GVL_MaintainLaser.q_bShutoffLatch := GVL_MaintainLaser.q_bShutoffLatch
	OR GVL_MaintainLaser.i_bShutoff
	OR NOT bSwitchboxStatusOk;
		
FOR nIter := 1 TO GVL_TransportTubes.NUM_TRANSPORT_TUBES DO
	eTT := GVL_TransportTubes.aTubes[nIter];
	fbTT REF= F_GetTransportTube(eTT);
	
	(* Disable Laser Ok signal if transport tube or switchbox is in bad state *)
	IF GVL_MaintainLaser.q_bShutoffLatch
	OR NOT F_VerifyTransportTubeStatuses(stExpStatus := stExpTTStatus,
		eTransportTube := eTT,
		stStatusOp := stTTOp, 
		bEnforce := FALSE)
	THEN // System status is not ok. Disable laser Ok signal
		fbTT.M_SetLaserOk(FALSE);
	END_IF
END_FOR

END_PROGRAM

// ---- POUs/Operations/MaintainLaser/FB_SwitchboxIonPumpFailure.TcPOU
(* Called to attempt to keep the laser on as long as safely possible in the event of an Ion Pump failure *)
FUNCTION_BLOCK FB_SwitchboxIonPumpFailure EXTENDS FB_MaintainLaserOperation
VAR_INPUT
END_VAR
VAR_OUTPUT
END_VAR
VAR
	fbVentSwitchbox: FB_VentSwitchbox;
END_VAR

SUPER^(iq_sMessageBuffer := iq_sMessageBuffer);

CASE eStep OF
E_OpStep.IDLE: // Do nothing

E_OpStep.START: // Turn on roughing pump
	M_RunTimeoutTimer(PUMP_TIMEOUT);
	M_SetMessage('Turning on roughing pump');
	
	GVL_BTS_VAC.fb_PP_PTM.M_Run(TRUE);
	
	IF GVL_BTS_VAC.fb_PP_PTM.iq_stPTM.eState = E_PumpState.pumpRUNNING THEN
		M_ResetTimeoutTimer();
		M_SetMessage('Turning off pumping station ion pump');
		eStep := E_OpStep.BOIP_TURN_OFF_ION_PUMP;
	END_IF
	
E_OpStep.BOIP_TURN_OFF_ION_PUMP:
	M_RunTimeoutTimer(PUMP_TIMEOUT);
	GVL_BTS_VAC.fb_PP_PIP.M_Run(FALSE);
	
	IF NOT GVL_BTS_VAC.fb_PP_PIP.i_xSP_DI THEN
		M_ResetTimeoutTimer();
		IF ABS(GVL_BTS_VAC.fb_PP_GPI_1.PG.rPRESS - GVL_BTS_VAC.fb_DP_GPI.PG.rPRESS) < 1E-4 THEN
			M_SetMessage('Opening pump station valve');
			eStep := E_OpStep.BOIP_OPEN_SB_VALVE;
		ELSE
			M_SetMessage('Unable to maintain vacuum');
			M_ShutdownLaser();
			eStep := E_OpStep.BOIP_VENT_SB;
		END_IF
	END_IF
	
E_OpStep.BOIP_OPEN_SB_VALVE:
	M_RunTimeoutTimer(VALVE_TIMEOUT);
	GVL_BTS_VAC.fb_PP_VGC.M_Set_OPN_SW(TRUE);
	
	IF GVL_BTS_VAC.fb_PP_VGC.M_IsOpen() THEN
		M_ResetTimeoutTimer();
		M_SetMessage('Maintaining vacuum');
		eStep := E_OpStep.BOIP_HOLD;
	END_IF
	
E_OpStep.BOIP_HOLD:
	// Hold vacuum as long as possible.
	IF GVL_BTS_VAC.fb_DP_GCC.IG.rPRESS > 1E-4 THEN
		// Shutdown laser
		M_ShutdownLaser();
		M_SetMessage('Vacuum lost. Closing transport tubes');
		eStep := E_OpStep.BOIP_CLOSE_TRANSPORT_TUBE_VALVES;
	END_IF

E_OpStep.BOIP_CLOSE_TRANSPORT_TUBE_VALVES:
	M_RunTimeoutTimer(VALVE_TIMEOUT);
	M_CloseAllTransportTubeValves();
	
	IF M_AllTransportTubeValvesClosed() THEN
		M_ResetTimeoutTimer();
		M_SetMessage('Closing switchbox valve');
		eStep := E_OpStep.BOIP_CLOSE_SB_VALVE;
	END_IF
	
E_OpStep.BOIP_CLOSE_SB_VALVE:
	M_RunTimeoutTimer(VALVE_TIMEOUT);
	GVL_BTS_VAC.fb_PP_VGC.M_Set_OPN_SW(FALSE);
	
	IF GVL_BTS_VAC.fb_PP_VGC.M_IsClosed() THEN
		M_ResetTimeoutTimer();
		M_SetMessage('Turning off switchbox pumps');
		eStep := E_OpStep.BOIP_TURN_OFF_PUMPS;
	END_IF

E_OpStep.BOIP_TURN_OFF_PUMPS:
	M_RunTimeoutTimer(PUMP_TIMEOUT);
	GVL_BTS_VAC.fb_PP_PTM.M_Run(FALSE);
	GVL_BTS_VAC.fb_PP_PMF.M_Run(FALSE);

	IF GVL_BTS_VAC.fb_PP_PTM.iq_stPTM.eState = E_PumpState.pumpSTOPPED AND GVL_BTS_VAC.fb_PP_PMF.q_stPump.eState = E_PumpState.pumpSTOPPED THEN
		M_ResetTimeoutTimer();
		M_SetMessage('Closing pump station valves');
		eStep := E_OpStep.BOIP_CLOSE_PP_VALVES;
	END_IF

E_OpStep.BOIP_CLOSE_PP_VALVES:
	M_RunTimeoutTimer(VALVE_TIMEOUT);
	GVL_BTS_VAC.fb_PP_VRC_1.M_Set_OPN_SW(FALSE);
	GVL_BTS_VAC.fb_PP_VRC_2.M_Set_OPN_SW(FALSE);
	
	IF GVL_BTS_VAC.fb_PP_VRC_1.iq_stValve.eState = E_ValvePositionState.CLOSED AND GVL_BTS_VAC.fb_PP_VRC_2.iq_stValve.eState = E_ValvePositionState.CLOSED THEN
		M_ResetTimeoutTimer();
		M_SetMessage('Venting switchbox');
		eStep := E_OpStep.BOIP_VENT_SB;	
	END_IF
	
E_OpStep.BOIP_VENT_SB:
	M_DeferCancel(TRUE);
	fbVentSwitchbox(i_bExecute := TRUE,
		i_bCancel := i_bCancel,
		iq_sMessageBuffer := iq_sMessageBuffer);
		
	IF fbVentSwitchbox.q_bError THEN
		M_DeferCancel(FALSE);
		M_FatalError('Error while venting switchbox');
	ELSIF NOT fbVentSwitchbox.q_bBusy THEN
		M_DeferCancel(FALSE);
		M_Finish();
	END_IF
	
ELSE
	M_FatalError('Operation is in invalid state');
END_CASE

END_FUNCTION_BLOCK

// ---- POUs/Operations/Abstracts/FB_MaintainLaserOperation.TcPOU
FUNCTION_BLOCK FB_MaintainLaserOperation EXTENDS FB_Operation
VAR_INPUT
END_VAR
VAR_OUTPUT
	q_bShutdownLaser : BOOL;
END_VAR
VAR
END_VAR

// Let FB_Operation do its thing 
SUPER^(iq_sMessageBuffer := iq_sMessageBuffer);

METHOD PROTECTED M_AllTransportTubeValvesClosed : BOOL
VAR_INPUT
END_VAR
VAR
	nIter : UINT;
	eTT : T_TransportTube;
	fbTT : REFERENCE TO FB_TransportTube;
END_VAR
M_AllTransportTubeValvesClosed := TRUE;

FOR nIter := 1 TO GVL_TransportTubes.NUM_TRANSPORT_TUBES DO
	eTT := GVL_TransportTubes.aTubes[nIter];
	fbTT REF= F_GetTransportTube(eTT);

	IF NOT fbTT.q_stConfig.stDevices.refGateValve.M_IsClosed() THEN
		M_AllTransportTubeValvesClosed := FALSE;
		RETURN;
	END_IF
END_FOR
END_METHOD

METHOD PROTECTED M_CloseAllTransportTubeValves
VAR_INPUT
END_VAR
VAR
	nIter : UINT;
	eTT : T_TransportTube;
	fbTT : REFERENCE TO FB_TransportTube;
END_VAR
FOR nIter := 1 TO GVL_TransportTubes.NUM_TRANSPORT_TUBES DO
	eTT := GVL_TransportTubes.aTubes[nIter];
	fbTT REF= F_GetTransportTube(eTT);

	fbTT.q_stConfig.stDevices.refGateValve.M_Set_OPN_SW(FALSE);
END_FOR
END_METHOD

METHOD PROTECTED M_FatalError
VAR_INPUT
	i_ErrorMessage : STRING;
END_VAR
SUPER^.M_FatalError(i_ErrorMessage);
M_ShutdownLaser();
END_METHOD

METHOD PUBLIC M_ResetError
VAR_INPUT
END_VAR
SUPER^.M_ResetError();
q_bShutdownLaser := FALSE;
END_METHOD

METHOD PROTECTED M_ShutdownLaser
VAR_INPUT
END_VAR
q_bShutdownLaser := TRUE;
END_METHOD

END_FUNCTION_BLOCK

// ---- POUs/Operations/MaintainLaser/FB_SwitchboxRoughingOrTurboPumpFailure.TcPOU
FUNCTION_BLOCK FB_SwitchboxRoughingOrTurboPumpFailure EXTENDS FB_MaintainLaserOperation
VAR_INPUT
END_VAR
VAR_OUTPUT
END_VAR
VAR
	fbVentSwitchbox: FB_VentSwitchbox;
END_VAR

SUPER^(iq_sMessageBuffer := iq_sMessageBuffer);

CASE eStep OF
E_OpStep.IDLE: // Do nothing

E_OpStep.START:
	M_RunTimeoutTimer(VALVE_TIMEOUT);
	GVL_BTS_VAC.fb_PP_VGC.M_Set_OPN_SW(FALSE);
	M_SetMessage('Closing switchbox valve');
	
	IF GVL_BTS_VAC.fb_PP_VGC.M_IsClosed() THEN
		M_ResetTimeoutTimer();
		IF GVL_BTS_VAC.fb_DP_GCC.IG.rPRESS < 1E-3 THEN
			M_SetMessage('Turn on ion pump');
			eStep := E_OpStep.BOPL_TURN_ON_ION_PUMP;
		ELSE
			M_SetMessage('Unable to maintain vacuum');
			M_ShutdownLaser();
			eStep := E_OpStep.BOPL_VENT_SB;
		END_IF
	END_IF

E_OpStep.BOPL_TURN_ON_ION_PUMP:
	M_RunTimeoutTimer(PUMP_TIMEOUT);
	GVL_BTS_VAC.fb_PP_PIP.M_Run(TRUE);
	
	IF NOT GVL_BTS_VAC.fb_PP_PIP.i_xSP_DI THEN
		M_ResetTimeoutTimer();
		M_SetMessage('Closing pumping station valves');
		eStep := E_OpStep.BOPL_CLOSE_PP_VALVES;
	END_IF
	
E_OpStep.BOPL_CLOSE_PP_VALVES:
	M_RunTimeoutTimer(VALVE_TIMEOUT);
	GVL_BTS_VAC.fb_PP_VRC_1.M_Set_OPN_SW(FALSE);
	GVL_BTS_VAC.fb_PP_VRC_2.M_Set_OPN_SW(FALSE);
	
	IF GVL_BTS_VAC.fb_PP_VRC_1.iq_stValve.eState = E_ValvePositionState.CLOSED AND GVL_BTS_VAC.fb_PP_VRC_2.iq_stValve.eState = E_ValvePositionState.CLOSED THEN
		M_ResetTimeoutTimer();
		M_SetMessage('Turning off pumping station pumps');
		eStep := E_OpStep.BOPL_TURN_OFF_PP_PUMPS;
	END_IF
	
E_OpStep.BOPL_TURN_OFF_PP_PUMPS:
	M_RunTimeoutTimer(PUMP_TIMEOUT);
	GVL_BTS_VAC.fb_PP_PTM.M_Run(FALSE);
	GVL_BTS_VAC.fb_PP_PMF.M_Run(FALSE);
	
	IF GVL_BTS_VAC.fb_PP_PTM.iq_stPTM.eState = E_PumpState.pumpSTOPPED AND GVL_BTS_VAC.fb_PP_PMF.q_stPump.eState = E_PumpState.pumpSTOPPED THEN
		M_ResetTimeoutTimer();
		M_SetMessage('Maintaining vacuum');
		eStep := E_OpStep.BOPL_HOLD;
	END_IF

E_OpStep.BOPL_HOLD:
	// Hold vacuum as long as possible.
	IF GVL_BTS_VAC.fb_DP_GCC.IG.rPRESS > 1E-4  THEN
		M_ShutdownLaser();
		M_SetMessage('Vacuum lost. Closing transport tubes');
		eStep := E_OpStep.BOPL_CLOSE_TRANSPORT_TUBE_VALVES;
	END_IF

E_OpStep.BOPL_CLOSE_TRANSPORT_TUBE_VALVES:
	M_RunTimeoutTimer(VALVE_TIMEOUT);
	M_CloseAllTransportTubeValves();
	
	IF M_AllTransportTubeValvesClosed() THEN
		M_ResetTimeoutTimer();
		M_SetMessage('Closing switchbox valve');
		eStep := E_OpStep.BOPL_VENT_SB;
	END_IF
	
E_OpStep.BOPL_VENT_SB:
	M_DeferCancel(TRUE);
	fbVentSwitchbox(i_bExecute := TRUE,
		i_bCancel := i_bCancel,
		iq_sMessageBuffer := iq_sMessageBuffer);
		
	IF fbVentSwitchbox.q_bError THEN
		M_DeferCancel(FALSE);
		M_FatalError('Error while venting switchbox');
	ELSIF NOT fbVentSwitchbox.q_bBusy THEN
		M_DeferCancel(FALSE);
		M_Finish();
	END_IF
	
ELSE
	M_FatalError('Operation is in invalid state');
END_CASE

END_FUNCTION_BLOCK

// ---- POUs/Operations/FB_OpenTransportTube.TcPOU
FUNCTION_BLOCK FB_OpenTransportTube EXTENDS FB_TTOperation
VAR
	fbPumpSwitchbox : FB_PumpSwitchbox;
	fbPumpTransportTube : FB_PumpTransportTube;
END_VAR

(*
SUPER^(iq_sMessageBuffer := iq_sMessageBuffer);

CASE eStep OF
E_OpStep.IDLE: // Do nothing

E_OpStep.START: // Verify system status	
	M_SetMessage('Verifying System Status');
	
	IF GVL_BTS_VAC.fb_DP_GCC.IG.rPRESS <= 1E-5 AND fbTT.q_stConfig.stDevices.refColdCathode.IG.rPRESS <= 1E-5 THEN 
		// System status check passed
		M_SetMessage('Opening gate valve');
		eStep := E_OpStep.OTT_OPEN_VALVE;
	// If either the switchbox or transport tube are not at base pressure, pump down the higher one
	ELSIF GVL_BTS_VAC.fb_DP_GCC.IG.rPRESS > fbTT.q_stConfig.stDevices.refColdCathode.IG.rPRESS THEN
		// Pump down switchbox
		M_SetMessage('Pumping switchbox');
		eStep := E_OpStep.OTT_RUN_PSB;
	ELSE // Pump down transport tube
		M_SetMessage('Pumping transport tube');
		eStep := E_OpStep.OTT_RUN_PTT;
	END_IF
	
E_OpStep.OTT_RUN_PSB: // Pump down switchbox
	M_DeferCancel(TRUE); // Make sure pump switchbox cancels before this operation does
	fbPumpSwitchbox(i_bExecute := TRUE,
		i_bCancel := i_bCancel,
		iq_sMessageBuffer := iq_sMessageBuffer);
		
	IF fbPumpSwitchbox.q_bError THEN
		M_DeferCancel(FALSE);
		M_FatalError('Error while pumping switchbox');
	ELSIF NOT fbPumpSwitchbox.q_bBusy THEN
		M_DeferCancel(FALSE);
		M_SetMessage('Retrying open transport tube');
		eStep := E_OpStep.START;
	END_IF
	
E_OpStep.OTT_RUN_PTT: // Pump transport tube
	M_DeferCancel(TRUE); // Make sure pump transport tube cancels before this operation does
	fbPumpTransportTube(i_bExecute := TRUE,
		i_bCancel := i_bCancel,
		iq_sMessageBuffer := iq_sMessageBuffer,
		i_eTransportTube := eTT);
		
	IF fbPumpTransportTube.q_bError THEN
		M_DeferCancel(FALSE);
		M_FatalError('Error while pumping transport tube');
	ELSIF NOT fbPumpTransportTube.q_bBusy THEN
		M_DeferCancel(FALSE);
		M_SetMessage('Retrying open transport tube');
		eStep := E_OpStep.START;
	END_IF
	
E_OpStep.OTT_OPEN_VALVE:
	M_RunTimeoutTimer(VALVE_TIMEOUT);
	
	// Open the gate valve
	fbTT.q_stConfig.stDevices.refGateValve.M_Set_OPN_SW(TRUE);
	
	// Once the gate valve is open, finish the operation
	IF fbTT.q_stConfig.stDevices.refGateValve.M_IsOpen() THEN
		M_ResetTimeoutTimer();
		M_Finish();
	END_IF
	
ELSE
	M_FatalError('Operation is in invalid state');
END_CASE
*)

END_FUNCTION_BLOCK

// ---- POUs/SystemStatusChecks/TransportTubes/F_GetTransportTubeStatuses.TcPOU
FUNCTION F_GetTransportTubeStatuses : ST_TransportTubeStatuses
VAR_INPUT
	eTransportTube : T_TransportTube;
END_VAR
VAR
	fbTT : REFERENCE TO FB_TransportTube;
	stStatus : ST_TransportTubeStatuses := ();
END_VAR

fbTT REF= F_GetTransportTube(eTransportTube);

stStatus.bIonPumpOn := fbTT.q_stConfig.stDevices.refIonPump.q_xHVEna_DO;
stStatus.bGateValveOpen := fbTT.q_stConfig.stDevices.refGateValve.M_IsOpen();
stStatus.fPiraniVal := fbTT.q_stConfig.stDevices.refPiraniGauge.PG.rPRESS;
stStatus.fColdCathodeVal := fbTT.q_stConfig.stDevices.refColdCathode.IG.rPRESS;

F_GetTransportTubeStatuses := stStatus;

END_FUNCTION

// ---- POUs/SystemStatusChecks/TransportTubes/F_SetTransportTubeStatuses.TcPOU
FUNCTION F_SetTransportTubeStatuses : BOOL
VAR_INPUT
	eTransportTube : T_TransportTube;
	stExpStatus : ST_TransportTubeStatuses;
	stStatusOp : ST_TransportTubeOps;
END_VAR
VAR
	fbTT : REFERENCE TO FB_TransportTube;
END_VAR

fbTT REF= F_GetTransportTube(eTransportTube);

IF NOT stStatusOp.bIonPumpIgnore THEN
	fbTT.q_stConfig.stDevices.refIonPump.M_Run(stExpStatus.bIonPumpOn);
END_IF
IF NOT stStatusOp.bGateValveIgnore THEN
	fbTT.q_stConfig.stDevices.refGateValve.M_Set_OPN_SW(stExpStatus.bGateValveOpen);
END_IF

END_FUNCTION
